INTERFACE I_Error EXTENDS I_Serializable, I_Disposable

PROPERTY ErrorType : T_MAXSTRING
GET
END_GET
END_PROPERTY

METHOD PUBLIC IsSameAs : BOOL
VAR_INPUT
	Error : I_Error;
END_VAR
END_METHOD

PROPERTY Message : T_MAXSTRING
GET
END_GET
END_PROPERTY

END_INTERFACE

(* stored: Version 1.1.0.1, ProductVersion 3.1.4024.12
   Itf I_Error: Id {039ad3bf-854e-4ff6-9567-e14fd8d09ff8}
   Property ErrorType: Id {c7f19ad6-32d2-0df7-0743-297efaa340a3}
   Get Get: Id {6c1aedeb-67d1-04eb-0630-eeedbbe111e7}
   Method IsSameAs: Id {81bd842e-8f00-08d7-203c-5ecdb55e1c31}
   Property Message: Id {3cfa7994-3809-44a2-babb-d6291d35c9f9}
   Get Get: Id {e87612e7-bf66-45b2-81e9-c318f4256621} *)
